Staubli VAL3: stop.pgx

program stop()
        begin
          resetMotion()
          disablePower()
        end
